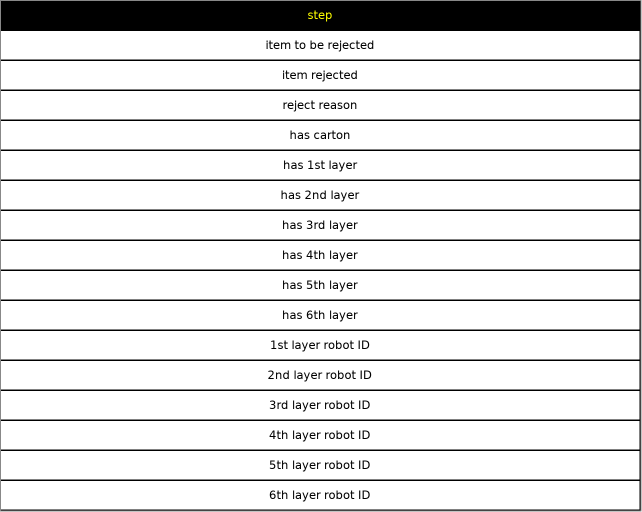
VISUALIZATION CARTON_FILLING_SHIFT_ELEMENT_DESCRIPTION  // 642x512
    Rectangle (0,0 640x30), "step"
    Rectangle (0,30 640x30), "item to be rejected"
    Rectangle (0,90 640x30), "reject reason"
    Rectangle (0,120 640x30), "has carton"
    Rectangle (0,150 640x30), "has 1st layer"
    Rectangle (0,60 640x30), "item rejected"
    Rectangle (0,180 640x30), "has 2nd layer"
    Rectangle (0,210 640x30), "has 3rd layer"
    Rectangle (0,240 640x30), "has 4th layer"
    Rectangle (0,270 640x30), "has 5th layer"
    Rectangle (0,300 640x30), "has 6th layer"
    Rectangle (0,330 640x30), "1st layer robot ID"
    Rectangle (0,360 640x30), "2nd layer robot ID"
    Rectangle (0,390 640x30), "3rd layer robot ID"
    Rectangle (0,420 640x30), "4th layer robot ID"
    Rectangle (0,450 640x30), "5th layer robot ID"
    Rectangle (0,480 640x30), "6th layer robot ID"
END_VISUALIZATION

(* stored: Version 1.1.0.1, ProductVersion 3.1.4024.3
   Visu CARTON_FILLING_SHIFT_ELEMENT_DESCRIPTION: Id {aa78a8b9-f50c-460d-84cd-7a8599d37f9f} *)
